TYPE DUT_SERVER_PARAMETERINPUTARRAY :
STRUCT
	ParameterInput0: DUT_PARAMETER_INPUT;
	ParameterInput1: DUT_PARAMETER_INPUT;
	ParameterInput2: DUT_PARAMETER_INPUT;
	ParameterInput3: DUT_PARAMETER_INPUT;
	ParameterInput4: DUT_PARAMETER_INPUT;
	ParameterInput5: DUT_PARAMETER_INPUT;
END_STRUCT
END_TYPE

(* stored: Version 1.1.0.1, ProductVersion 3.1.0.25
   DUT DUT_SERVER_PARAMETERINPUTARRAY: Id {1504cd0c-9764-466f-b682-b1de8b428888} *)
